// TIA Portal V17 export
// export: Created 2024-01-30T08:54:10.0026641Z, ExportSetting WithDefaults, DisplayName Totally Integrated Automation Portal, DisplayVersion V17 Update 6, DisplayName TIA Portal Openness, DisplayVersion V17 Update 6, DisplayName TIA Portal Version Control Interface, DisplayVersion V17, DisplayName STEP 7 Professional, DisplayVersion V17 Update 6, DisplayName STEP 7 Safety, DisplayVersion V17 Update 6, DisplayName WinCC Advanced, DisplayVersion V17 Update 6
VAR_GLOBAL   // PLC tag table "LJ_X8000"
   PLC_to_LJ_X8000bits AT %Q2.0 : "UDT_PLC --> LJ_X8000_Bits";
   PLC_to_LJ_X8000bytes AT %Q27.0 : "UDT_PLC --> LJ_X8000_Bytes";
   LJ_X8000_to_PLCbits AT %I22.0 : "UDT_LJ_X8000 --> PLC_Bits";
   LJ_X8000_to_PLCbytes AT %I34.0 : "UDT_LJ_X8000 --> PLC_Bytes";
   NewVariables AT %I98.0 : "UDT_LJ_X8000 --> PLC_Bytes";
END_VAR
